TYPE ST_IdentityOUT1 :
STRUCT
	ID	:STRING;
	ReadQuality:STRING;
END_STRUCT
END_TYPE

(* stored: Version 1.1.0.1, ProductVersion 3.1.4024.13
   DUT ST_IdentityOUT1: Id {72a3e9b0-bd7b-44e6-8016-b5a6c9a86d0d} *)
